Fanuc KAREL source: NC0027.KL

-- PROVISIONAL review KL for V770-1; original PC SHA256 600b0563a3ba21f315cfd7f3c78fc507f88492308e5573fd5aca7977d7802ce0
-- Incomplete behavior may be omitted. Consult companion uncertainty JSON. Do not deploy.
PROGRAM NC0027
%NOLOCKGROUP
-- UNRESOLVED_LOCAL_POOL 1 cells at code offset 3; source declarations unknown
-- DIRECT_LOCAL_WORD_ACCESS alone does not prove INTEGER, REAL, or BOOLEAN
BEGIN
  -- UNRESOLVED_PC offsets 0-8; opcodes 2B,2C,7B
  -- UNRESOLVED_PC offsets 13-20; opcodes 9D,23
  -- UNRESOLVED_PC offsets 25-42; opcodes 21,40,41,42
  -- UNRESOLVED_PC offsets 47-64; opcodes 21,40,41,42
  -- UNRESOLVED_PC offsets 69-86; opcodes 21,40,41,42
  -- UNRESOLVED_PC offsets 91-108; opcodes 21,40,41,42
  -- UNRESOLVED_PC offsets 113-130; opcodes 21,40,41,42
  -- UNRESOLVED_PC offsets 135-152; opcodes 21,40,41,42
  -- UNRESOLVED_PC offsets 157-174; opcodes 21,40,41,42
  -- UNRESOLVED_PC offsets 179-196; opcodes 21,40,41,42
  -- UNRESOLVED_PC offsets 201-218; opcodes 21,40,41,42
  -- UNRESOLVED_PC offsets 223-240; opcodes 21,40,41,42
  -- UNRESOLVED_PC offsets 245-275; opcodes 21,9D,52,23,7A,40,41,42
  -- UNRESOLVED_PC offsets 280-304; opcodes 21,2E,52,23,7A,43
  -- UNRESOLVED_PC offsets 309-327; opcodes 21,2E,52,23
  -- UNRESOLVED_PC offsets 332-348; opcodes 7A,40,41,42
  -- UNRESOLVED_PC offsets 353-377; opcodes 21,2E,52,23,7A,43
  -- UNRESOLVED_PC offsets 382-400; opcodes 21,2E,52,23
  -- UNRESOLVED_PC offsets 405-421; opcodes 7A,40,41,42
  -- UNRESOLVED_PC offsets 426-450; opcodes 21,2E,52,23,7A,43
  -- UNRESOLVED_PC offsets 455-473; opcodes 21,2E,52,23
  -- UNRESOLVED_PC offsets 478-494; opcodes 7A,40,41,42
  -- UNRESOLVED_PC offsets 499-523; opcodes 21,2E,52,23,7A,43
  -- UNRESOLVED_PC offsets 528-546; opcodes 21,2E,52,23
  -- UNRESOLVED_PC offsets 551-567; opcodes 7A,40,41,42
  -- UNRESOLVED_PC offsets 572-596; opcodes 21,2E,52,23,7A,43
  -- UNRESOLVED_PC offsets 601-619; opcodes 21,2E,52,23
  -- UNRESOLVED_PC offsets 624-640; opcodes 7A,40,41,42
  -- UNRESOLVED_PC offsets 645-669; opcodes 21,2E,52,23,7A,43
  -- UNRESOLVED_PC offsets 674-692; opcodes 21,2E,52,23
  -- UNRESOLVED_PC offsets 697-713; opcodes 7A,40,41,42
  -- UNRESOLVED_PC offsets 718-742; opcodes 21,2E,52,23,7A,43
  -- UNRESOLVED_PC offsets 747-765; opcodes 21,2E,52,23
  -- UNRESOLVED_PC offsets 770-786; opcodes 7A,40,41,42
  -- UNRESOLVED_PC offsets 791-815; opcodes 21,2E,52,23,7A,43
  -- UNRESOLVED_PC offsets 820-838; opcodes 21,2E,52,23
  -- UNRESOLVED_PC offsets 843-859; opcodes 7A,40,41,42
  -- UNRESOLVED_PC offsets 864-888; opcodes 21,2E,52,23,7A,43
  -- UNRESOLVED_PC offsets 893-911; opcodes 21,2E,52,23
  -- UNRESOLVED_PC offsets 916-932; opcodes 7A,40,41,42
  -- UNRESOLVED_PC offsets 937-961; opcodes 21,2E,52,23,7A,43
  -- UNRESOLVED_PC offsets 966-984; opcodes 21,2E,52,23
  -- UNRESOLVED_PC offsets 994-998; opcodes 7F
  -- UNRESOLVED_PC offsets 1003-1007; opcodes 27,AA
  -- UNRESOLVED_PC offsets 1012-1016; opcodes 7F
END NC0027
